{attribute addProperty BoxType "AT2042-0250-0024"}
{attribute addProperty Id "A_0098_AT2025_5250_0019_AT2025_5250AT2025_3DCFC8D064080"}
{attribute addProperty CRC "451507384"}
{attribute addProperty SizeInBites "640"}
{attribute addProperty SizeInBytes "80"}
TYPE A_0046_AT2042_0250_0024_1AE974B8 EXTENDS AT2042_9506A482 :
STRUCT
	{attribute addProperty Name "A_0098_AT2025_5250_0019_AT2025_5250"}
	A_0098_AT2025_5250_0019_AT2025_5250 : AT2025_3DCFC8D0;
END_STRUCT
END_TYPE

(* stored: Version 1.2.0.0, ProductVersion 3.1.4024.9
   DUT A_0046_AT2042_0250_0024_1AE974B8: Id {beca63a0-6d96-449a-8ada-7d554e44119d} *)
